FUNCTION_BLOCK PackMLTestSuite EXTENDS TcUnit.FB_TestSuite
VAR
END_VAR

CheckBasicStateMachineCycle();

METHOD PUBLIC CheckBasicStateMachineCycle
VAR_INST
	state_machine : StateMachine<State.Idle>;
END_VAR
Test('CheckStateMachine');

AssertTrue(
	Condition := state_machine.IsIdle,
	Message := 'State machine is not in Idle state immediately after creation'
);

state_machine.Start();
AssertTrue(
	Condition := state_machine.IsStarting,
	Message := 'State machine is not in Starting state immediately after Start action'
);

state_machine.StateComplete();
AssertTrue(
	Condition := state_machine.IsExecuting,
	Message := 'State machine is not in Execute state immediately after Starting state complete'
);

state_machine.StateComplete();
AssertTrue(
	Condition := state_machine.IsCompleting,
	Message := 'State machine is not in Completing state immediately after Execute state complete'
);

state_machine.StateComplete();
AssertTrue(
	Condition := state_machine.IsCompleted,
	Message := 'State machine is not in Completed state immediately after Completing state complete'
);

state_machine.Reset();
AssertTrue(
	Condition := state_machine.IsResetting,
	Message := 'State machine is not in Resetting state immediately after Reset action'
);

state_machine.StateComplete();
AssertTrue(
	Condition := state_machine.IsIdle,
	Message := 'State machine is not in Idle state immediately after Resetting state complete'
);

Test_Finished();
END_METHOD

END_FUNCTION_BLOCK

(* stored: Version 1.1.0.1
   POU PackMLTestSuite: Id {a4e9f584-02fa-02ab-0aa2-33b7dba803f2}, SpecialFunc None
   Method CheckBasicStateMachineCycle: Id {bf387793-5f99-0aa2-3285-02bd6db473a3} *)
